% RSLogix 500 project segment_drum_volume.RSS, saved by version 8.30.00.16 %
PROJECT "UNTITLED"    % processor: Bul.1763 MicroLogix 1100 Series B %

PROGRAM FILES
  LAD 2   5 rungs

DATA FILES
  O0 OUTPUT  4 elements
  I1 INPUT  6 elements
  S2 STATUS  66 elements
  B3 BINARY  1 elements
  T4 TIMER  1 elements
  C5 COUNTER  1 elements
  R6 CONTROL  1 elements
  N7 INTEGER  3 elements
  F8 FLOAT  8 elements
  F10 SCAN_RSLTS  65 elements  % pass_areas %
  F11 SCAN_CHCKS  65 elements
  F12 SCAN_LVLS  65 elements
  F13 SCAN_SCANS  65 elements

LADDER 2
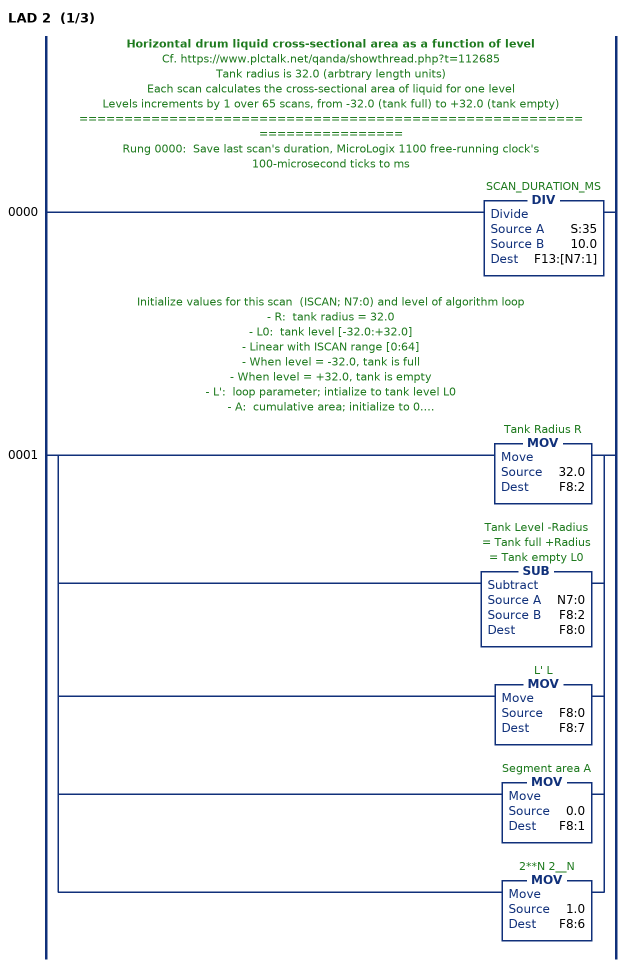
% Rung: 0 %
% TITLE: Horizontal drum liquid cross-sectional area as a function of level %
% Cf. https://www.plctalk.net/qanda/showthread.php?t=112685
% 
% Tank radius is 32.0 (arbtrary length units)
% Each scan calculates the cross-sectional area of liquid for one level
% Levels increments by 1 over 65 scans, from -32.0 (tank full) to +32.0 (tank empty)
% 
% ========================================================================
% Rung 0000:  Save last scan's duration, MicroLogix 1100 free-running clock's 100-microsecond ticks to ms %
SOR DIV S:35 10.0 F13:[N7:1] EOR
%   S:35  "Last 1 ms Scan Time" %
%   F13:[N7:1]  SCAN_DURATION_MS %
%   N7:1  LAST_ISCAN  "Last scan number" %
% Rung: 1 %
% Initialize values for this scan  (ISCAN; N7:0) and level of algorithm loop
% - R:  tank radius = 32.0
% - L0:  tank level [-32.0:+32.0]
%   - Linear with ISCAN range [0:64]
%   - When level = -32.0, tank is full
%   - When level = +32.0, tank is empty
% - L':  loop parameter; intialize to tank level L0
% - A:  cumulative area; initialize to 0.0
% - 2**N:  per-loop scale factor; initialize to 1.0 %
SOR BST MOV 32.0 F8:2 NXB SUB N7:0 F8:2 F8:0 NXB MOV F8:0 F8:7 NXB MOV 0.0 F8:1 NXB MOV 1.0 F8:6 BND EOR
%   F8:2  R  "Tank Radius" %
%   N7:0  ISCAN  "Scan number, [0:64]" %
%   F8:0  L0  "Tank Level -Radius = Tank full +Radius = Tank empty" %
%   F8:7  L  "L'" %
%   F8:1  A  "Segment area" %
%   F8:6  2__N  "2**N" %

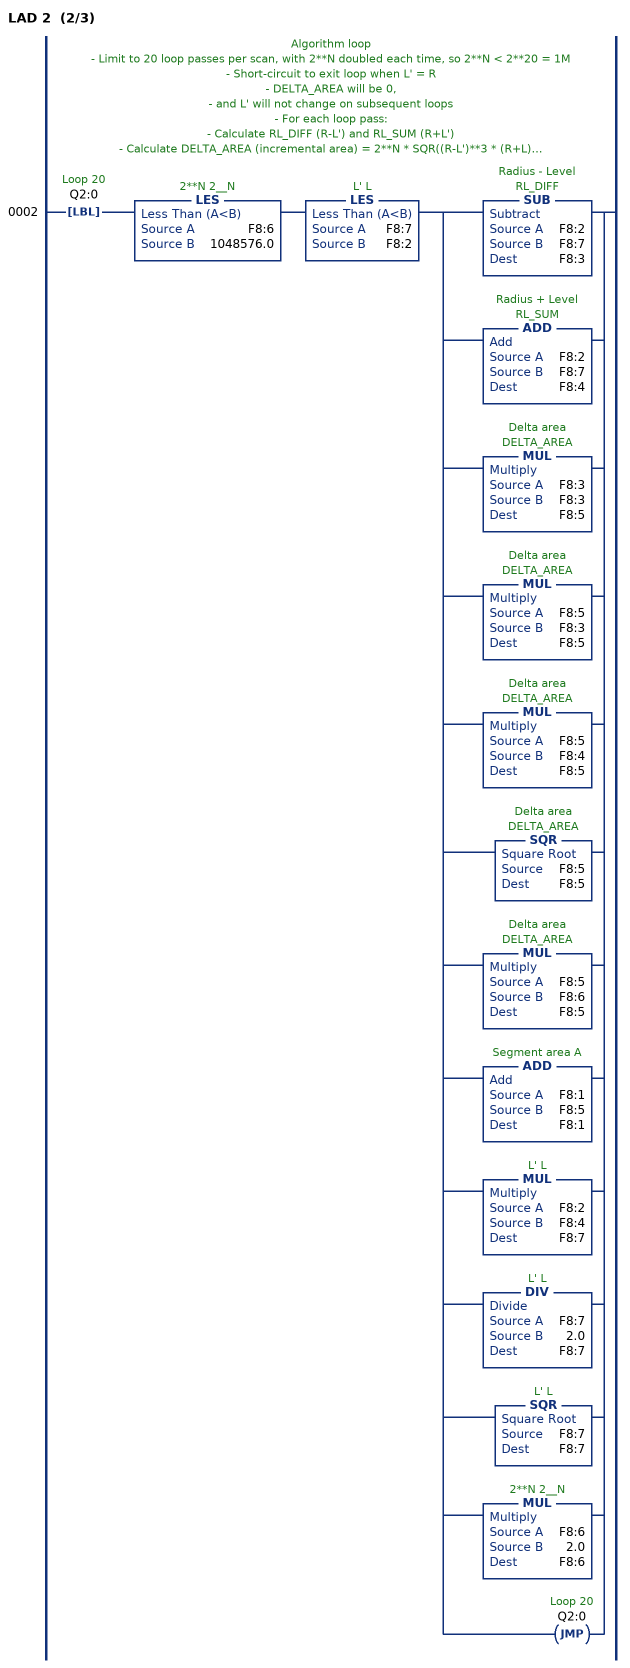
% Rung: 2 %
% Algorithm loop
% - Limit to 20 loop passes per scan, with 2**N doubled each time, so 2**N < 2**20 = 1M
%   - Short-circuit to exit loop when L' = R
%     - DELTA_AREA will be 0,
%     - and L' will not change on subsequent loops
% - For each loop pass:
%   - Calculate RL_DIFF (R-L') and RL_SUM (R+L')
%   - Calculate DELTA_AREA (incremental area) = 2**N * SQR((R-L')**3 * (R+L))
%   - Increment cumulative Area (A): A = A + DELTA_AREA
%   - Advance L' parameter for next loop pass:  L' = SQR(R * (R+L') / 2)
%   - Double 2**N factor
%   - Repeat loop %
SOR LBL Q2:0 LES F8:6 1048576.0 LES F8:7 F8:2 BST SUB F8:2 F8:7 F8:3 NXB ADD F8:2 F8:7 F8:4 NXB MUL F8:3 F8:3 F8:5 NXB MUL F8:5 F8:3 F8:5 NXB MUL F8:5 F8:4 F8:5 NXB SQR F8:5 F8:5 NXB MUL F8:5 F8:6 F8:5 NXB ADD F8:1 F8:5 F8:1 NXB MUL F8:2 F8:4 F8:7 NXB DIV F8:7 2.0 F8:7 NXB SQR F8:7 F8:7 NXB MUL F8:6 2.0 F8:6 NXB JMP Q2:0 BND EOR
%   Q2:0  "Loop 20" %
%   F8:6  2__N  "2**N" %
%   F8:7  L  "L'" %
%   F8:2  R  "Tank Radius" %
%   F8:3  RL_DIFF  "Radius - Level" %
%   F8:4  RL_SUM  "Radius + Level" %
%   F8:5  DELTA_AREA  "Delta area" %
%   F8:1  A  "Segment area" %

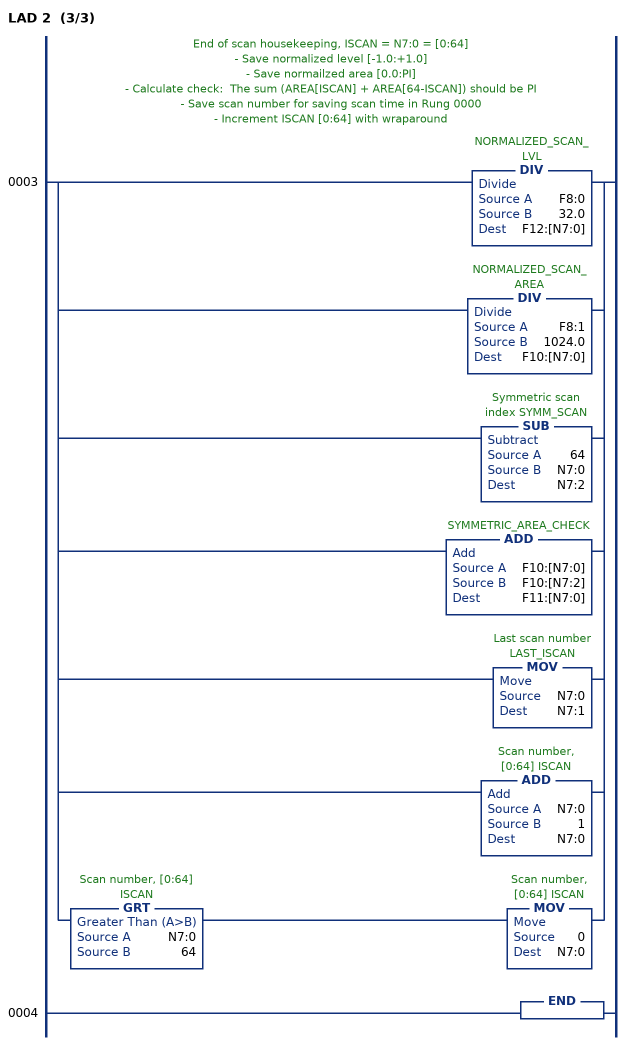
% Rung: 3 %
% End of scan housekeeping, ISCAN = N7:0 = [0:64]
% - Save normalized level [-1.0:+1.0]
% - Save normailzed area [0.0:PI]
% - Calculate check:  The sum (AREA[ISCAN] + AREA[64-ISCAN]) should be PI
% - Save scan number for saving scan time in Rung 0000
% - Increment ISCAN [0:64] with wraparound %
SOR BST DIV F8:0 32.0 F12:[N7:0] NXB DIV F8:1 1024.0 F10:[N7:0] NXB SUB 64 N7:0 N7:2 NXB ADD F10:[N7:0] F10:[N7:2] F11:[N7:0] NXB MOV N7:0 N7:1 NXB ADD N7:0 1 N7:0 NXB GRT N7:0 64 MOV 0 N7:0 BND EOR
%   F8:0  L0  "Tank Level -Radius = Tank full +Radius = Tank empty" %
%   F12:[N7:0]  NORMALIZED_SCAN_LVL %
%   N7:0  ISCAN  "Scan number, [0:64]" %
%   F8:1  A  "Segment area" %
%   F10:[N7:0]  NORMALIZED_SCAN_AREA %
%   N7:2  SYMM_SCAN  "Symmetric scan index" %
%   F10:[N7:2]  SYMMETRIC_SCAN_AREA %
%   F11:[N7:0]  SYMMETRIC_AREA_CHECK %
%   N7:1  LAST_ISCAN  "Last scan number" %
% Rung: 4 %
SOR END EOR

OTHER DOCUMENTED ADDRESSES
  F10:[N7:1]  NORMALIZED_SYMM_AREA
  N9:[N7:1]  "Last scan's duration"

DATA TABLE (non-zero values as saved)
DATA F8
% F8:0 % 5 0 32 0 0
